// Mitsubishi GX Works2 project: 231002-001- exercicios-3   PLC: Q03UDV

// global labels: Global1
VAR_GLOBAL
  Up_Down AT M34 : BOOL;
END_VAR

// task Task_01 (event TRUE, interval 0, priority 31): POU_01

PROGRAM POU_01
VAR
  CTD_1 : CTD;
  CTU_1 : CTU;
  meuc : CTU;
  novo : CTUD;
END_VAR
(* structured ladder/FBD written out as ST: instructions are called as NAME(EN, inputs, outputs); _pN, _eN, _tN stand for wires *)
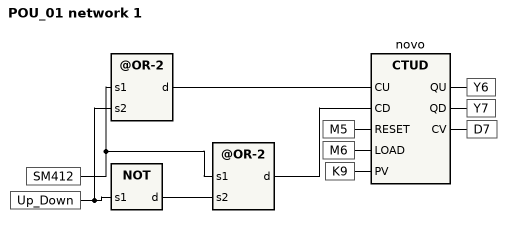
(* network 1 *)
novo(CU := @OR-2(SM412, Up_Down), CD := @OR-2(SM412, NOT(Up_Down)), RESET := M5, LOAD := M6, PV := K9, QU => Y6, QD => Y7, CV => D7);
END_PROGRAM
